// SIMATIC S7-200 project (STEP 7-Micro/WIN), CPU 226XM REL 01.22

SYMBOL_TABLE USER1
bezczynnosc_do_za_gorac M1.7     // w彻cz wiatrak
bezczynnosc_do_za_zimno M1.6     // w彻cz grzanie
ANDwb            M1.5     // wy彻czenie wiatraka
ANDgb            M1.4     // wy彻czenie grza砶i
RSwentylator     M1.3
RSgrzalka        M1.2
RSbezczynnosc    M1.1
ANDgrzalka       M0.6
bezczynnosc      M0.5
ANDwentylator    M0.7
T_z_sub_h        VW130
T_z_add_h        VW120
h                VW110
T_ge_T_z         M0.2
T_z_ge_T         M0.1
h_count          C1
T_z              VW100
T_z_count        C0
T                AIW8
END_SYMBOL_TABLE

ORGANIZATION_BLOCK MAIN:OB1
TITLE=PROGRAM COMMENTS
BEGIN
Network 1
LD     SM0.0
CALL   ASI0_CTRL:SBR1, VB48
Network 2
// AND wentylator  (dodac T> T_z + h)
LD     M0.0
A      RSbezczynnosc:M1.1
=      ANDwentylator:M0.7
Network 3
// AND grzalka (dodac T_z - h > T)
LD     M0.0
A      RSbezczynnosc:M1.1
=      ANDgrzalka:M0.6
Network 4
// AND grzalka -> bezczynnosc (dodac T >= T_z)
LD     M0.0
A      RSgrzalka:M1.2
=      ANDgb:M1.4
Network 5
// AND wentylator -> bezczynnosc (dodac T <= T_z)
LD     M0.0
A      RSwentylator:M1.3
=      ANDwb:M1.5
Network 6
LD     SM0.1
O      ANDgb:M1.4
O      ANDwb:M1.5
LD     ANDwentylator:M0.7
O      ANDgrzalka:M0.6
NOT
LPS
A      Q0.3
=      Q0.3
LPP
ALD
O      Q0.3
=      Q0.3
=      RSbezczynnosc:M1.1
=      Q0.0
Network 7
// w彻cz wiatrak
LD     ANDwentylator:M0.7
LD     ANDwb:M1.5
NOT
LPS
A      Q0.1
=      Q0.1
LPP
ALD
O      Q0.1
=      Q0.1
=      RSwentylator:M1.3
=      Q0.0
Network 8
// w彻cz grzanie
LD     ANDgrzalka:M0.6
LD     ANDgb:M1.4
NOT
LPS
A      Q0.2
=      Q0.2
LPP
ALD
O      Q0.2
=      Q0.2
=      RSgrzalka:M1.2
=      Q0.0
END_ORGANIZATION_BLOCK

// SBR1: protected block, not included

// SBR2: protected block, not included

// SBR3: protected block, not included
